{attribute 'GeneratedUsingTerminal: KL2641-0001'}
{attribute addProperty BoxType "KL2641-0001"}
{attribute addProperty Description ""}
{attribute addProperty Physics ""}
{attribute addProperty Id "Channel_1AT %Q*Channel_BF3661CD0"}
{attribute addProperty CRC "2942934076"}
{attribute addProperty Size "0"}
TYPE KL_AF699C3C :
STRUCT
	{attribute addProperty Name "Channel_1"}
	Channel_1 : Channel_BF3661CD;
END_STRUCT
END_TYPE

(* stored: Version 1.2.0.0, ProductVersion 3.1.4024.9
   DUT KL_AF699C3C: Id {08d48d85-6945-4ff0-9ee3-51206f1e7aaa} *)
